FUNCTION_BLOCK FB_TimersTEST
VAR_INPUT
	bStartTON	: BOOL;
	bStartTOF	: BOOL;
	tTime		: TIME;
END_VAR

VAR_IN_OUT	
	tTON			: TON;
	tTOF			: TOF;
END_VAR

VAR_OUTPUT
	tTON_Q		: BOOL;
	tTOF_Q		: BOOL;
END_VAR
VAR
	tPTton			: TIME;
	tPTtof			: TIME;
	
END_VAR


tPTtof := tTime;
tPTton := tTime;

tTON(IN := bStartTON, PT := tPTton, Q => tTON_Q);
tTOF(IN := bStartTOF, PT := tPTtof, Q => tTOF_Q);

END_FUNCTION_BLOCK

(* stored: Version 1.1.0.1
   POU FB_TimersTEST: Id {170a98dc-72aa-41ee-b056-1f311026d0ec}, SpecialFunc None *)
